TYPE ST_EmonioP3DefaultParameters :
STRUCT
	fCalorificValue : REAL := 11.49;
END_STRUCT
END_TYPE

(* stored: Version 1.1.0.1, ProductVersion 3.1.4024.10
   DUT ST_EmonioP3DefaultParameters: Id {9cca4352-ee73-4052-8640-058793b09631} *)
